// TIA Portal V17 export
// export: Created 2024-08-29T18:23:51.02087Z, ExportSetting WithDefaults, DisplayName Totally Integrated Automation Portal, DisplayVersion V17 Update 7, DisplayName TIA Portal Openness, DisplayVersion V17 Update 7, DisplayName TIA Portal Version Control Interface, DisplayVersion V17, DisplayName SINAMICS Startdrive Advanced, DisplayVersion V17 SP2, DisplayName SINAMICS Startdrive G110M, G120, G120C, G120D, G120P, G115D, DisplayVersion V17 SP2, DisplayName SINAMICS Startdrive G130, G150, S120, S150, SINAMICS MV, S210, DisplayVersion V17 SP2, DisplayName STEP 7 Professional, DisplayVersion V17 Update 7, DisplayName STEP 7 Safety, DisplayVersion V17 Update 6, DisplayName WinCC Advanced / Unified PC, DisplayVersion V17 Update 7
TYPE "udtButtons"
// stored: IsFailsafeCompliant false
   STRUCT
      bReq : Bool;
      bP : Bool;
      bTGG : Bool;
      bCmd : Bool;
      bAkn : Bool;
      b1 : Bool;
      b2 : Bool;
      b3 : Bool;
   END_STRUCT;
END_TYPE
